Omron CX-Programmer project NewProject (CX-Programmer 9.61)

# PLC NewPLC1: CP1E N30

## Global symbols (name address type ; comment)
0.00 BOOL  ; PB1
100 CHANNEL  ; $?St$Bk?_#[10] / $?St$Bk?_#[10]
100.00 BOOL  ; Pilot lamp
101 CHANNEL  ; 100
T000 BOOL  ; Timer 1

## Program NewProgram1 (cyclic task 0)

### Section Section1

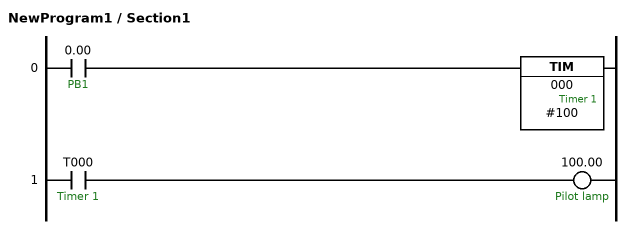
; rung 0
LD 0.00  ; PB1
TIM 000 #100  ; Timer 1
; rung 1
LD T000  ; Timer 1
OUT 100.00  ; Pilot lamp

### Section END
; rung 0
END(001)